(* CODESYS project CtaVisMouseEvent_1.0.0.0.library
   Description: Visu Mouse Event Library der CTA
   Version: 1.0.0.0
   Title: CtaVisMouseEvent
   Author: SIS
   LanguageModelAttribute: qualified-access-only
   DocFormat: reStructuredText
   Placeholder: CtaVisMouseEvent
   DefaultNamespace: CtaVisMouseEvent
   CompiledLibraryCompatibilityVersion: CODESYS V3.5 SP16 Patch 3
   Company: CTA

Project tree, tasks and I/O mapping:
  libraries: VisuElemBase, * (System); CtaSysEvent, 1.0.0.0 (CTA)
  40 Visualizations/
  30 Program Organization Units/
    function block FB_MOUSE_EVENT_MANAGER [ST]: ADD_MOUSE_EVENT_LISTNER, REM_MOUSE_EVENT_NODE, FB_INIT, HandleMouseBtnEvent, HandleMouseMoveEvent, metStartDone, metPrepeareStop, metCyclicCall, proDenyStop, proIsRegistred
    function block FB_MOUSE_EVENT_NODE [ST]: BIG_SYBIL, SELF, LOW_SYBIL, REGISTER, FB_EXIT, UNREGISTER, FB_INIT, HandleMouseBtnEvent, HandleMouseMoveEvent
  00000000-0000-0000-0000-000000000000|D:\CoDeSys\LibrariesV3\trunk\Intern\CAA\CAA Template\3.4.0.0 draft\Placeholder.xml
  00000000-0000-0000-0000-000000000000|D:\CoDeSys\LibrariesV3\trunk\Intern\CAA\CAA Template\3.2.0.3 draft\Prefix.pdf
  00000000-0000-0000-0000-000000000000|D:\CoDeSys\LibrariesV3\trunk\Intern\CAA\CAA Template\3.5.2.0 draft\Placeholder.xml
  20 Structs/
    data type enEventType
  50 Images/
  10 Documenation/
    global variables VersionHistory
    global variables readMe
  21 Interface/
    interface ITF_MOUSE_EVENT_NODE: BIG_SYBIL, LOW_SYBIL, SELF, HandleMouseBtnEvent, HandleMouseMoveEvent
  11 Library Parameter/
  12 Konstanten/
  60 Textlisten/
  13 Globale Variablen/
    global variables GVL_MOUSE_EVENT
  5ce3da45-db07-42e7-a21c-a00fff4ed8f6|Icons\alert.svg
  5ce3da45-db07-42e7-a21c-a00fff4ed8f6|Icons\arrow-down.svg
  5ce3da45-db07-42e7-a21c-a00fff4ed8f6|Icons\arrow-down_square.svg
  5ce3da45-db07-42e7-a21c-a00fff4ed8f6|Icons\arrow-left_solo_black.svg
  5ce3da45-db07-42e7-a21c-a00fff4ed8f6|Icons\arrow-right_solo_black.svg
  5ce3da45-db07-42e7-a21c-a00fff4ed8f6|Icons\arrow-up.svg
  5ce3da45-db07-42e7-a21c-a00fff4ed8f6|Icons\calendar-range.svg
  5ce3da45-db07-42e7-a21c-a00fff4ed8f6|Icons\check.svg
  5ce3da45-db07-42e7-a21c-a00fff4ed8f6|Icons\clock-outline.svg
  5ce3da45-db07-42e7-a21c-a00fff4ed8f6|Icons\close_solo_black.svg
  5ce3da45-db07-42e7-a21c-a00fff4ed8f6|Icons\CtaInfo.svg
  5ce3da45-db07-42e7-a21c-a00fff4ed8f6|Icons\database_black.svg
  5ce3da45-db07-42e7-a21c-a00fff4ed8f6|Icons\delete_solo_black.svg
  5ce3da45-db07-42e7-a21c-a00fff4ed8f6|Icons\engine.svg
  5ce3da45-db07-42e7-a21c-a00fff4ed8f6|Icons\front_hand_Black.svg
  5ce3da45-db07-42e7-a21c-a00fff4ed8f6|Icons\front_hand_Yellow_Off.svg
  5ce3da45-db07-42e7-a21c-a00fff4ed8f6|Icons\gear.svg
  5ce3da45-db07-42e7-a21c-a00fff4ed8f6|Icons\home.svg
  5ce3da45-db07-42e7-a21c-a00fff4ed8f6|Icons\information-variant.svg
  5ce3da45-db07-42e7-a21c-a00fff4ed8f6|Icons\lightning-bolt-circle.svg
  5ce3da45-db07-42e7-a21c-a00fff4ed8f6|Icons\message.svg
  5ce3da45-db07-42e7-a21c-a00fff4ed8f6|Icons\message-alert-variant.svg
  5ce3da45-db07-42e7-a21c-a00fff4ed8f6|Icons\minus_solo_black.svg
  5ce3da45-db07-42e7-a21c-a00fff4ed8f6|Icons\plus_solo_black.svg
  5ce3da45-db07-42e7-a21c-a00fff4ed8f6|Icons\power_solo_black.svg
  5ce3da45-db07-42e7-a21c-a00fff4ed8f6|Icons\refresh_solo_black.svg
  5ce3da45-db07-42e7-a21c-a00fff4ed8f6|Icons\SearchFilter.svg
  5ce3da45-db07-42e7-a21c-a00fff4ed8f6|Icons\signal-celular-alt.svg
  5ce3da45-db07-42e7-a21c-a00fff4ed8f6|Icons\toggle-switch.svg
  5ce3da45-db07-42e7-a21c-a00fff4ed8f6|Icons\Modbus_Organization_Logo.svg
  5ce3da45-db07-42e7-a21c-a00fff4ed8f6|Icons\CheckboxUnchecked_withe.svg
  5ce3da45-db07-42e7-a21c-a00fff4ed8f6|Icons\lock_open_black.svg
  5ce3da45-db07-42e7-a21c-a00fff4ed8f6|Icons\check_green.svg
  5ce3da45-db07-42e7-a21c-a00fff4ed8f6|Icons\filter_black.svg
  5ce3da45-db07-42e7-a21c-a00fff4ed8f6|Icons\CtaLogo.png
  5ce3da45-db07-42e7-a21c-a00fff4ed8f6|Icons\Grafana_Logo.svg
  5ce3da45-db07-42e7-a21c-a00fff4ed8f6|Icons\hourglass_top.svg
  text list GlobalTextList
*)

// 20 Structs/enEventType
{attribute 'qualified_only'}
{attribute 'strict'}
TYPE enEventType :
(
	MOUSE_DOWN	:=	0,
	MOUSE_UP	:=	1,
	MOUSE_KLIK	:=	2
);
END_TYPE;

// 10 Documenation/VersionHistory
(* 

.. image:: ../../Images/CTA_Logo.jpg
   :align: right
   :width: 15% 

**Vorlage**   


============ =========== =========== ============================================
**Date**     **Version** **Author**  **Change**
------------ ----------- ----------- --------------------------------------------
04.03.2021   0.0.0.0     SIS         Vorlage erstellt

============ =========== =========== ============================================


*)
VAR_GLOBAL
    stInfo : STRING:= '0.0.0.0, Vorlage, CTA';
END_VAR

// 10 Documenation/readMe
(*

**ReadMe**
 
|	**Empfehlung**
|
|	Der FB_MOUSE_EVENT_NODE dient der verarbeitung spezifischer Mouse events.
|     
*)

VAR_GLOBAL
    xReadMeDone              :   BOOL;
END_VAR

// 13 Globale Variablen/GVL_MOUSE_EVENT
{attribute 'qualified_only'}
{attribute 'linkalways'}
{attribute 'global_init_slot' := '40010'}
VAR_GLOBAL
	FB_MOUSE_EVENT_MANAGER	:	FB_MOUSE_EVENT_MANAGER;
END_VAR

// 30 Program Organization Units/FB_MOUSE_EVENT_MANAGER
{attribute 'hide'}
FUNCTION_BLOCK FB_MOUSE_EVENT_MANAGER IMPLEMENTS VisuElemBase.IMouseEventHandler , CtaSysEvent.ITF_APPEVENT
VAR_INPUT
END_VAR
VAR_OUTPUT
END_VAR
VAR
	(* Event Nodes *)
	_BASE_EVENT_NODE	:	ITF_MOUSE_EVENT_NODE;
	_TEMP_REG_NODE		:	ITF_MOUSE_EVENT_NODE;
	_EVENT_TYPE			:	enEventType;
	_xIsRegistred		:	BOOL;
END_VAR

METHOD ADD_MOUSE_EVENT_LISTNER
VAR_INPUT
	ITF_MOUSE_EVENT_NODE_IN	:	ITF_MOUSE_EVENT_NODE;
END_VAR
(* Check Base Node *)
IF __QUERYINTERFACE(_BASE_EVENT_NODE,_BASE_EVENT_NODE) THEN
	(* Check Temp Node *)
	IF __QUERYINTERFACE(_TEMP_REG_NODE,_TEMP_REG_NODE) THEN
		(* Set Low Sybill *)
		_TEMP_REG_NODE.LOW_SYBIL := ITF_MOUSE_EVENT_NODE_IN;
		(* Set New Temp Node *)
		_TEMP_REG_NODE := ITF_MOUSE_EVENT_NODE_IN;
	ELSE
		(* Set Temp Node *)
		_TEMP_REG_NODE 				:= ITF_MOUSE_EVENT_NODE_IN;
		(* Set Base Node Low Sybil *)
		_BASE_EVENT_NODE.LOW_SYBIL 	:= ITF_MOUSE_EVENT_NODE_IN;
	END_IF;		
ELSE
	(* Set Base Node *)
	_BASE_EVENT_NODE := ITF_MOUSE_EVENT_NODE_IN;
END_IF
END_METHOD

METHOD REM_MOUSE_EVENT_NODE 
VAR_INPUT
	ITF_MOUSE_EVENT_NODE_IN	:	ITF_MOUSE_EVENT_NODE;
END_VAR
VAR
	_ITF_BIG_SYBIL	:	ITF_MOUSE_EVENT_NODE;
	_ITF_LOW_SYBIL	:	ITF_MOUSE_EVENT_NODE;
END_VAR
(* Check if Node is valid *)
IF __QUERYINTERFACE(ITF_MOUSE_EVENT_NODE_IN,ITF_MOUSE_EVENT_NODE_IN) THEN
	(* Get Big Sybil *)
	_ITF_BIG_SYBIL := ITF_MOUSE_EVENT_NODE_IN.BIG_SYBIL;
	(* Get Low Sybil *)
	_ITF_LOW_SYBIL := ITF_MOUSE_EVENT_NODE_IN.LOW_SYBIL;
	(* Check if Node is Base Node *)
	IF ITF_MOUSE_EVENT_NODE_IN = _BASE_EVENT_NODE THEN
		(* Check if Low Sybil is valid *)
		IF __QUERYINTERFACE(_ITF_LOW_SYBIL,_ITF_LOW_SYBIL) THEN
			(* Set Low Sybil as Base Node *)
			_BASE_EVENT_NODE := _ITF_LOW_SYBIL;
		ELSE
			(* Set Base Node to 0 *)
			_BASE_EVENT_NODE := 0;
		END_IF;
	END_IF;
	(* Check if Big Sybil is Valid *)
	IF __QUERYINTERFACE(_ITF_BIG_SYBIL,_ITF_BIG_SYBIL) THEN
		(* Add Low Sybill as Low Sybill of Big Sybill *)
		_ITF_BIG_SYBIL.LOW_SYBIL := _ITF_LOW_SYBIL;
	END_IF;
	(* Check if Low Sybil is Valid *)
	IF __QUERYINTERFACE(_ITF_LOW_SYBIL,_ITF_LOW_SYBIL) THEN
		(* Add Big Sybill as Big Sybill of Low Sybill *)
		_ITF_LOW_SYBIL.BIG_SYBIL := _ITF_BIG_SYBIL;
	END_IF;
	(* Delete Sybils of Node *)
	ITF_MOUSE_EVENT_NODE_IN.BIG_SYBIL := 0;
	ITF_MOUSE_EVENT_NODE_IN.LOW_SYBIL := 0;
END_IF;
END_METHOD

//FB_Init ist immer implizit verfügbar und wird primär für die Initialisierung verwendet.
//Der Rückgabewert wird nicht ausgewertet. Für gezielte Einflussnahme können Sie
//die Methoden explizit deklarieren und darin mit dem Standard-Initialisierungscode 
//zusätzlichen Code bereitstellen. Sie können den Rückgabewert auswerten.
METHOD FB_Init: BOOL
VAR_INPUT    
bInitRetains: BOOL; // TRUE: Die Retain-Variablen werden initialisiert (Reset warm / Reset kalt)    
bInCopyCode: BOOL;  // TRUE: Die Instanz wird danach in den Kopiercode kopiert (Online-Change)
END_VAR
IF NOT bInCopyCode THEN
	CtaSysEvent.fcRegistry(THIS^);
	VisuElemBase.Visu_Globals.g_VisuEventManager.SetMouseEventHandler(THIS^);
END_IF;
END_METHOD

(* This method will be called when a mouse button is pressed. 
 RETURN: 
 TRUE - When the handler has handled this event and it should not be handled by someone else
 FALSE - When the event is not handled by this handler*)
METHOD HandleMouseBtnEvent : BOOL
VAR_INPUT
	(* The event type. The value is true if a mouse button was released.*)
	bMouseUpEvent	: BOOL;
	(* Information about the button that was pressed or released. At the moment this
 value is not yet used and will always have the value 0!*)
	btMouseBtn	: BYTE;
	(* The position where the mouse event was raised. The coordinates of this point are relative to the 
 currently active toplevel visualization, even when best fit is activated.  *)
	ptMouse	: VisuElemBase.VisuStructPoint;
	(* A pointer to the client structure were the event occurred.*)
	pClient	: POINTER TO VisuElemBase.VisuStructClientData;

END_VAR
VAR
	_TEMP_EVENT_NODE	:	ITF_MOUSE_EVENT_NODE;
END_VAR
(* Check Mouse Down Event *)
IF NOT bMouseUpEvent THEN
	(* Set Mouse Down Event *)
	_EVENT_TYPE := enEventType.MOUSE_DOWN;
(* Check if Mouse Up Event after Mouse Down event *)
ELSIF bMouseUpEvent AND _EVENT_TYPE = enEventType.MOUSE_DOWN THEN
	(* Set Mouse Up Event *)
	_EVENT_TYPE := enEventType.MOUSE_UP;
(* Check if Mouse Klick event is send *)	
ELSIF bMouseUpEvent AND _EVENT_TYPE = enEventType.MOUSE_UP THEN
	(* Set Mouse Klick Event *)
	_EVENT_TYPE := enEventType.MOUSE_KLIK;
END_IF;
(* Check Base Node *)
IF __QUERYINTERFACE(_BASE_EVENT_NODE,_TEMP_EVENT_NODE) THEN
	REPEAT
		(* Check Temp Node *)
		IF __QUERYINTERFACE(_TEMP_EVENT_NODE,_TEMP_EVENT_NODE) THEN
			(* Call Mouse Event *)
			_TEMP_EVENT_NODE.HandleMouseBtnEvent(bMouseUpEvent,btMouseBtn,ptMouse,pClient,_EVENT_TYPE);
			(* Get Low Sybill *)
			_TEMP_EVENT_NODE := _TEMP_EVENT_NODE.LOW_SYBIL;
		END_IF;
	(* End Repeat if no more Nodes *)
	UNTIL _TEMP_EVENT_NODE = 0
	END_REPEAT
END_IF;
HandleMouseBtnEvent := FALSE;
END_METHOD

(* This method will be called when the mouse was moved. 
 RETURN: 
 TRUE - When the handler has handled this event and it should not be handled by someone else
 FALSE - When the event is not handled by this handler*)
METHOD HandleMouseMoveEvent : BOOL
VAR_INPUT
	(* The position where the mouse was moved to. The coordinates of this point are relative to the 
 currently active toplevel visualization, even when best fit is activated.  *)
	ptMouse	: VisuElemBase.VisuStructPoint;
	(* A pointer to the client structure were the event occurred.*)
	pClient	: POINTER TO VisuElemBase.VisuStructClientData;
END_VAR
VAR
	_TEMP_EVENT_NODE	:	ITF_MOUSE_EVENT_NODE;
END_VAR
(* Check Base Node *)
IF __QUERYINTERFACE(_BASE_EVENT_NODE,_TEMP_EVENT_NODE) THEN
	REPEAT
		(* Check Temp Node *)
		IF __QUERYINTERFACE(_TEMP_EVENT_NODE,_TEMP_EVENT_NODE) THEN
			(* Call Mouse Event *)
			_TEMP_EVENT_NODE.HandleMouseMoveEvent(ptMouse,pClient);
			(* Get Low Sybill *)
			_TEMP_EVENT_NODE := _TEMP_EVENT_NODE.LOW_SYBIL;
		END_IF;
	(* End Repeat if no more Nodes *)
	UNTIL _TEMP_EVENT_NODE = 0
	END_REPEAT
END_IF;
END_METHOD

METHOD metStartDone : BOOL
RETURN;
END_METHOD

METHOD metPrepeareStop : BOOL
RETURN;
END_METHOD

METHOD metCyclicCall : BOOL
VisuElemBase.Visu_Globals.g_VisuEventManager.SetMouseEventHandler(THIS^);
END_METHOD

PROPERTY proDenyStop : BOOL
GET
proDenystop := FALSE;
END_GET
END_PROPERTY

PROPERTY proIsRegistred : BOOL
GET
proIsRegistred := _xIsRegistred;
END_GET
SET
_xIsRegistred := proIsRegistred;
END_SET
END_PROPERTY

END_FUNCTION_BLOCK

// 21 Interface/ITF_MOUSE_EVENT_NODE
INTERFACE ITF_MOUSE_EVENT_NODE EXTENDS __SYSTEM.IQueryInterface

PROPERTY BIG_SYBIL : ITF_MOUSE_EVENT_NODE
GET
END_GET
SET
END_SET
END_PROPERTY

PROPERTY LOW_SYBIL : ITF_MOUSE_EVENT_NODE
SET
END_SET
GET
END_GET
END_PROPERTY

PROPERTY SELF : ITF_MOUSE_EVENT_NODE
GET
END_GET
END_PROPERTY

(* This method will be called when a mouse button is pressed. 
 RETURN: 
 TRUE - When the handler has handled this event and it should not be handled by someone else
 FALSE - When the event is not handled by this handler*)
METHOD HandleMouseBtnEvent : BOOL
VAR_INPUT
	(* The event type. The value is true if a mouse button was released.*)
	bMouseUpEvent	: BOOL;
	(* Information about the button that was pressed or released. At the moment this
 value is not yet used and will always have the value 0!*)
	btMouseBtn	: BYTE;
	(* The position where the mouse event was raised. The coordinates of this point are relative to the 
 currently active toplevel visualization, even when best fit is activated.  *)
	ptMouse	: VisuElemBase.VisuStructPoint;
	(* A pointer to the client structure were the event occurred.*)
	pClient	: POINTER TO VisuElemBase.VisuStructClientData;
	EVENT_TYPE	:	enEventType;
END_VAR
END_METHOD

(* This method will be called when the mouse was moved. 
 RETURN: 
 TRUE - When the handler has handled this event and it should not be handled by someone else
 FALSE - When the event is not handled by this handler*)
METHOD HandleMouseMoveEvent : BOOL
VAR_INPUT
	(* The position where the mouse was moved to. The coordinates of this point are relative to the 
 currently active toplevel visualization, even when best fit is activated.  *)
	ptMouse	: VisuElemBase.VisuStructPoint;
	(* A pointer to the client structure were the event occurred.*)
	pClient	: POINTER TO VisuElemBase.VisuStructClientData;
END_VAR
END_METHOD

END_INTERFACE

// 30 Program Organization Units/FB_MOUSE_EVENT_NODE
FUNCTION_BLOCK FB_MOUSE_EVENT_NODE IMPLEMENTS ITF_MOUSE_EVENT_NODE
VAR_INPUT
END_VAR
VAR_OUTPUT
END_VAR
VAR
	_ITF_BIG_SYBIL	:	ITF_MOUSE_EVENT_NODE;
	_ITF_LOW_SYBIL	:	ITF_MOUSE_EVENT_NODE;
END_VAR

{attribute 'estimated-stack-usage' := '104'}
PROPERTY FINAL BIG_SYBIL : ITF_MOUSE_EVENT_NODE
GET
BIG_SYBIL := _ITF_BIG_SYBIL;
END_GET
SET
_ITF_BIG_SYBIL := BIG_SYBIL;
IF __QUERYINTERFACE(_ITF_BIG_SYBIL,_ITF_BIG_SYBIL) THEN
	IF _ITF_BIG_SYBIL.LOW_SYBIL <> SELF THEN
		_ITF_BIG_SYBIL.LOW_SYBIL := THIS^;
	END_IF;
END_IF;
END_SET
END_PROPERTY

PROPERTY FINAL SELF : ITF_MOUSE_EVENT_NODE
GET
SELF := THIS^;
END_GET
END_PROPERTY

{attribute 'estimated-stack-usage' := '104'}
PROPERTY FINAL LOW_SYBIL : ITF_MOUSE_EVENT_NODE
GET
LOW_SYBIL := _ITF_LOW_SYBIL;
END_GET
SET
_ITF_LOW_SYBIL := LOW_SYBIL;
IF __QUERYINTERFACE(_ITF_LOW_SYBIL,_ITF_LOW_SYBIL) THEN
	IF _ITF_LOW_SYBIL.BIG_SYBIL <> SELF THEN
		_ITF_LOW_SYBIL.BIG_SYBIL := THIS^;
	END_IF;
END_IF;
END_SET
END_PROPERTY

METHOD FINAL REGISTER 
VAR_INPUT
END_VAR
(* Add Mouse Event Listner Node *)
GVL_MOUSE_EVENT.FB_MOUSE_EVENT_MANAGER.ADD_MOUSE_EVENT_LISTNER(THIS^);
END_METHOD

//FB_Exit muss explizit implementiert werden. Wenn es eine Implementierung gibt, dann wird 
//die Methode aufgerufen, bevor die Steuerung den Code der Funktionsbaustein-Instanz entfernt
//(impliziter Aufruf. Der Rückgabewert wird nicht ausgewertet.
METHOD FB_Exit: BOOL
VAR_INPUT    
bInCopyCode: BOOL;  // TRUE: Die Exit-Methode wird aufgerufen, um die Instanz zu verlassen, die hinterher kopiert wird Online-Change).  
END_VAR
(* Unregister on Exit *)
UNREGISTER();
END_METHOD

METHOD FINAL UNREGISTER 
VAR_INPUT
END_VAR
(* Remove Node *)
GVL_MOUSE_EVENT.FB_MOUSE_EVENT_MANAGER.REM_MOUSE_EVENT_NODE(THIS^);
END_METHOD

//FB_Init ist immer implizit verfügbar und wird primär für die Initialisierung verwendet.
//Der Rückgabewert wird nicht ausgewertet. Für gezielte Einflussnahme können Sie
//die Methoden explizit deklarieren und darin mit dem Standard-Initialisierungscode 
//zusätzlichen Code bereitstellen. Sie können den Rückgabewert auswerten.
METHOD FB_Init: BOOL
VAR_INPUT    
bInitRetains: BOOL; // TRUE: Die Retain-Variablen werden initialisiert (Reset warm / Reset kalt)    
bInCopyCode: BOOL;  // TRUE: Die Instanz wird danach in den Kopiercode kopiert (Online-Change)
END_VAR
(* Unregister *)
UNREGISTER();
(* Register *)
REGISTER();
END_METHOD

(* This method will be called when a mouse button is pressed. 
 RETURN: 
 TRUE - When the handler has handled this event and it should not be handled by someone else
 FALSE - When the event is not handled by this handler*)
METHOD HandleMouseBtnEvent : BOOL
VAR_INPUT
	(* The event type. The value is true if a mouse button was released.*)
	bMouseUpEvent	: BOOL;
	(* Information about the button that was pressed or released. At the moment this
 value is not yet used and will always have the value 0!*)
	btMouseBtn	: BYTE;
	(* The position where the mouse event was raised. The coordinates of this point are relative to the 
 currently active toplevel visualization, even when best fit is activated.  *)
	ptMouse	: VisuElemBase.VisuStructPoint;
	(* A pointer to the client structure were the event occurred.*)
	pClient	: POINTER TO VisuElemBase.VisuStructClientData;
	EVENT_TYPE	:	enEventType;
END_VAR
END_METHOD

(* This method will be called when the mouse was moved. 
 RETURN: 
 TRUE - When the handler has handled this event and it should not be handled by someone else
 FALSE - When the event is not handled by this handler*)
METHOD HandleMouseMoveEvent : BOOL
VAR_INPUT
	(* The position where the mouse was moved to. The coordinates of this point are relative to the 
 currently active toplevel visualization, even when best fit is activated.  *)
	ptMouse	: VisuElemBase.VisuStructPoint;
	(* A pointer to the client structure were the event occurred.*)
	pClient	: POINTER TO VisuElemBase.VisuStructClientData;
END_VAR
END_METHOD

END_FUNCTION_BLOCK
